Staubli VAL3: stop.pgx

public program stop()
  local num l_i
begin
  call StopAll()


end
